// TIA Portal V17 export
// export: Created 2022-07-20T07:01:28.7712866Z, ExportSetting WithDefaults, DisplayName Totally Integrated Automation Portal, DisplayVersion V17, DisplayName TIA Portal Openness, DisplayVersion V17, DisplayName TIA Portal Version Control Interface, DisplayVersion V17, DisplayName SINAMICS Startdrive Advanced, DisplayVersion V17, DisplayName SINAMICS Startdrive G130, G150, S120, S150, SINAMICS MV, S210, DisplayVersion V17, DisplayName SINAMICS Startdrive G110M, G120, G120C, G120D, G120P, G115D, DisplayVersion V17, DisplayName STEP 7 Professional, DisplayVersion V17, DisplayName STEP 7 Safety, DisplayVersion V17, DisplayName WinCC Advanced, DisplayVersion V17
FUNCTION_BLOCK "FB10251_IfmDV2510"   // FB10251, LAD
{ S7_Optimized_Access := 'TRUE' }
VERSION : 0.1
// stored: AutoNumber false, IsIECCheckEnabled false, IsRetainMemResEnabled false, MemoryReserve 100, SetENOAutomatically false, UDAEnableTagReadback false
   VAR_INPUT
      Segment1_Color : Byte;
      Segment1_Frequency : Byte;
      Segment2_Color : Byte;
      Segment2_Frequency : Byte;
      Segment3_Color : Byte;
      Segment3_Frequency : Byte;
      Segment4_Color : Byte;
      Segment4_Frequency : Byte;
      Segment5_Color : Byte;
      Segment5_Frequency : Byte;
      BuzerActivation : Bool;
      BuzerStyle : Byte;
   END_VAR
   VAR_IN_OUT
      ProcessDataWord_0 : Word;
      ProcessDataWord_2 : Word;
      ProcessDataWord_4 : Word;
   END_VAR
BEGIN

REGION Network 1 (SCL): Segment 1
   #ProcessDataWord_4 := 0;
   #ProcessDataWord_4.%B0 := #Segment1_Color OR #Segment1_Frequency;
   #ProcessDataWord_4.%B1 := #Segment2_Color OR #Segment2_Frequency;
END_REGION

REGION Network 2 (SCL): Segment 2
   #ProcessDataWord_2 := 0;
   #ProcessDataWord_2.%B0 := #Segment3_Color OR #Segment3_Frequency;
   #ProcessDataWord_2.%B1 := #Segment4_Color OR #Segment4_Frequency;
END_REGION

REGION Network 3 (SCL): Segment 2
   #ProcessDataWord_0 := 0;
   #ProcessDataWord_0.%B0 := #Segment5_Color OR #Segment5_Frequency;
   #ProcessDataWord_0.%B1 := #BuzerStyle;
   #ProcessDataWord_0.%X8 := #BuzerActivation;
END_REGION
END_FUNCTION_BLOCK
